{attribute 'GeneratedUsingTerminal: EJ2522-0000-0022'}
{attribute addProperty BoxType "EJ2522-0000-0022"}
{attribute addProperty Id "StatusAT %I*Status_70E023F86Counter_valueAT %I*UDINT4"}
{attribute addProperty CRC "2837785672"}
{attribute addProperty Size "10"}
TYPE ENC_Status_Channel_A9252C48 :
STRUCT
	{attribute addProperty Name "Status"}
	Status AT %I* : Status_70E023F8;
	{attribute addProperty Name "Counter_value"}
	Counter_value AT %I* : UDINT;
END_STRUCT
END_TYPE

(* stored: Version 1.2.0.0, ProductVersion 3.1.4024.9
   DUT ENC_Status_Channel_A9252C48: Id {5027893c-1a73-4617-abed-dae2ed78c3fd} *)
